FUNCTION_BLOCK RunCommonRack EXTENDS RunUnitGeneric
VAR_INPUT
	isEject : BOOL; //link to coordinator
END_VAR
VAR_OUTPUT
END_VAR
VAR
	commEject AT%M* : BOOL; // link to HMI, one shot commnad	

	button : POINTER TO RunSignal ;
	fixer : POINTER TO RunCylinder;
	approx : POINTER TO RunSignal; // approx then lock
	
	signal : ProgrammedOutput;
	//---------------------------------
	//	Over Fieldbus linked with SCARA
	//---------------------------------
	rackReady AT%Q*: BOOL;
	rackEngaged AT%I*: BOOL;	

	items : ARRAY[0..4] OF defItem;
	
	//---------------------------------
	//	Internal
	//---------------------------------
	nCounter : INT;
END_VAR


//Control the working flow of rack

SUPER^();

CASE outputState OF
	//----------------
	//	Initialization
	//----------------
	eSpecialStates.INITIAL_BEGIN:	
		bSerialTransition := fixer^.Execute(eCylinderCommands.COMMAND_A); //release
		IF bSerialTransition THEN
			rackReady := FALSE; //signal clearing
		END_IF
	eSpecialStates.INITIAL_STATE_1:
		//wait until synchronized with SCARA
		IF NOT rackEngaged THEN
			NextState:=eSpecialStates.INITIAL_END;
		END_IF
	//-----------------
	//	Working
	//-----------------
	eSpecialStates.GENERIC_GROUP_START:
		//rack is empty
		bSerialTransition := fixer^.Execute(eCylinderCommands.COMMAND_A); //relase
		signal.Activate(2);//50% set light flicking
	16#1:
		bSerialTransition := approx^.debouncedOn; //wait until rack closed
	16#2:
		//confirmed by hanshaking
		bSerialTransition := button^.debouncedOn;
		signal.Activate(0);//set light constant on
	16#3:
		bSerialTransition := fixer^.Execute(eCylinderCommands.COMMAND_B); //lock
		IF bSerialTransition THEN
			rackReady := TRUE;
			
			isEject := FALSE; //reset
		END_IF
	16#4:
		//------------------------------------------------------------------
		//	Check if any item reached the bound. then set rackReady as false
		// or by external signal (manual or job stop)
		//------------------------------------------------------------------
		FOR nCounter := 0 TO 3 DO
			IF items[nCounter].Counter >= items[nCounter].CurrerntIndex THEN
				bSerialTransition := TRUE;
				
			END_IF
		END_FOR
		bSerialTransition := bSerialTransition OR isEject OR commEject OR button^.onTimeElapsed > T#2S;
		
		IF bSerialTransition THEN
			rackReady := FALSE; //released
		END_IF
	16#5:
		//wait until SCARA disengaged
		IF NOT rackEngaged THEN
			NextState := eSpecialStates.GENERIC_GROUP_START; //rewind
		END_IF
END_CASE

commEject := FALSE;

METHOD FB_init : BOOL
VAR_INPUT
	bInitRetains : BOOL; // if TRUE, the retain variables are initialized (warm start / cold start)
	bInCopyCode : BOOL;  // if TRUE, the instance afterwards gets moved into the copy code (online change)
	
	argParent : POINTER TO RunUnitGeneric;
	argSlotBase : POINTER TO RunMaterial;
	argSlotLast : POINTER TO RunMaterial;
	
	argButton : POINTER TO RunSignal ;
	argFixer : POINTER TO RunCylinder;
	argApprox : POINTER TO RunSignal; 
END_VAR
//initialize 
Parent := argParent;
SlotBase := argSlotBase;
SlotLast := argSlotLast;
//
IF bInitRetains THEN
	NextState := eSpecialStates.INITIAL_BEGIN;
END_IF

button :=argButton;
fixer :=argFixer;
approx :=argApprox;
END_METHOD

END_FUNCTION_BLOCK

(* stored: Version 1.1.0.1, ProductVersion 3.1.4024.0
   POU RunCommonRack: Id {eac928e2-459d-4027-a156-266e564c65fe}, SpecialFunc None
   Method FB_init: Id {cdcb6566-3495-422b-9f0f-68d1a83249c2} *)
